TYPE SafetyHydraulicsStatuses :
STRUCT
	///Is the safety in a healthy state? Good=RUN, Bad=safe stopped
	healthStatus: HealthStatus;
	///Is the safety busy?
	busyStatus: BusyStatus;
END_STRUCT
END_TYPE

(* stored: Version 1.1.0.1, ProductVersion 3.1.4019.2
   DUT SafetyHydraulicsStatuses: Id {e26f6990-81ab-4ffd-a18b-6e69ab932145} *)
